// TwinCAT 3 PLC project PLC
// ProgramVersion: 3.1.4024.0
// libraries:
//   Tc2_Standard, * (Beckhoff Automation GmbH)
//   Tc2_System, * (Beckhoff Automation GmbH)
//   Tc3_Module, * (Beckhoff Automation GmbH)
// project tree:
//   / PlcTask.TcTTO
//   POUs/ MAIN.TcPOU
// real-time tasks:
//   TASK PlcTask: cycle T#1ms, priority 20, ADS port 350
// I/O:
//   DEVICE Device 3 (EtherCAT), AmsNetId 172.18.136.151.4.1
//     Box 1 (EP9224-0023) [EP9224-0023 4Ch/4Ch enhanced Power Distribution for EtherCAT Box Modules]
//     Box 2 (EP4174-0002) [EP4174-0002 4Ch. Ana. Output +/-10V, 0-10V, 0/4-20mA configurable]
// variable links:
//   PLC/PLC Instance <-> Device 3 (EtherCAT)/Box 1 (EP9224-0023)
//     PlcTask Outputs/MAIN.bChangeDirectionSmartRoller_KISS <-> DPO Outputs Channel 1/Output Us
//     PlcTask Outputs/MAIN.bChangeDirectionSmartRoller_Velo <-> DPO Outputs Channel 4/Output Us
//     PlcTask Outputs/MAIN.bEnableControlViaFieldbus <-> DPO Outputs Device/Enable Control Via Fieldbus
//     PlcTask Outputs/MAIN.bEnableSmartRoller_KISS <-> DPO Outputs Channel 1/Output Up
//     PlcTask Outputs/MAIN.bEnableSmartRoller_Velo <-> DPO Outputs Channel 4/Output Up
//   PLC/PLC Instance <-> Device 3 (EtherCAT)/Box 2 (EP4174-0002)
//     PlcTask Outputs/MAIN.nAnalogOutput <-> AO Outputs Channel 4/Analog output

CONFIGURATION PLC
    RESOURCE PLC ON TwinCAT3
        TASK PlcTask(INTERVAL := T#1ms, PRIORITY := 20);
        PROGRAM MAIN WITH PlcTask : MAIN;
    END_RESOURCE
END_CONFIGURATION

// ---- POUs/MAIN.TcPOU
PROGRAM MAIN
VAR
	bEnableControlViaFieldbus 			AT%Q*:BOOL; 
	bEnableSmartRoller_KISS				AT%Q*:BOOL; 
	bChangeDirectionSmartRoller_KISS 	AT%Q*:BOOL; 
	
	bEnableSmartRoller_Velo				AT%Q*:BOOL;
	bChangeDirectionSmartRoller_Velo	AT%Q*:BOOL;
	nAnalogOutput						AT%Q*: INT;
	nMinThreshold						:INT:=10000;
	nMaxThreshold						:INT:=32767;
	bRampPos							:BOOL;
	bEnableAnalogBox_Up					AT%Q*:BOOL; 
	bEnableAnalogBox_Us					AT%Q*:BOOL; 
END_VAR

IF bEnableSmartRoller_Velo THEN
	nAnalogOutput:=LIMIT(nMinThreshold,SEL(bRampPos,nAnalogOutput-1,nAnalogOutput+1),nMaxThreshold);
	IF nAnalogOutput>=nMaxThreshold THEN
		bRampPos:=FALSE;
	ELSIF nAnalogOutput<=nMinThreshold THEN
		bRampPos:=TRUE;
	END_IF
ELSE 
	nAnalogOutput:=0;
END_IF
bEnableControlViaFieldbus:=TRUE;
bEnableAnalogBox_Up:=TRUE;
bEnableAnalogBox_Us:=TRUE;

END_PROGRAM
